INTERFACE IShelf EXTENDS __SYSTEM.IQueryInterface

METHOD getNextFreeSpace : IShelfElement
VAR_INPUT
END_VAR
END_METHOD

METHOD getNextOccupiedSpace : IShelfElement
VAR_INPUT
END_VAR
END_METHOD

METHOD getShelfSpaceByPartId : IShelfElement
VAR_INPUT
	partId: STRING(23);
END_VAR
END_METHOD

PROPERTY m : UINT
GET
END_GET
END_PROPERTY

PROPERTY n : UINT
GET
END_GET
END_PROPERTY

METHOD storePart : BOOL
VAR_INPUT
	element: IShelfElement;
END_VAR
END_METHOD

METHOD unloadNextPart : IPart
VAR_INPUT
END_VAR
END_METHOD

METHOD unloadPartById : BOOL
VAR_INPUT
	partId: STRING(23);
END_VAR
END_METHOD

END_INTERFACE

(* stored: Version 1.1.0.1
   Itf IShelf: Id {f284db6d-1392-46f6-b464-a9431fe4cffb}
   Method getNextFreeSpace: Id {a75db583-e457-4555-91ad-3b9d9b19f8d3}
   Method getNextOccupiedSpace: Id {0802cca4-3a95-41a2-9a25-2f55f921c8cd}
   Method getShelfSpaceByPartId: Id {8a7fb1d2-7c90-4ef1-be25-d9a367ccd3c7}
   Property m: Id {246d4f74-70c3-4d93-a509-1f242d621233}
   Get Get: Id {f37d521f-d346-4510-804a-419a5da9aae9}
   Property n: Id {0bda7b08-7783-443a-a2c9-3b0924b0433b}
   Get Get: Id {8b7a1fe1-fea6-4f44-9c7f-7321704bfbe5}
   Method storePart: Id {bf45d5a5-c04c-41d8-9b4c-21d3ef1d6150}
   Method unloadNextPart: Id {a07823c0-25d9-47b7-9924-4d72f5336bfb}
   Method unloadPartById: Id {b38da53a-8e36-43d8-b398-1d52ab51a0ae} *)
